// Library/Structures/WorkArea/RobotWorkArea
{attribute 'pack_mode' := '1'} 
// ------------------------------------------------------------------------- 
//  SRCI Robot Library                                                
// ------------------------------------------------------------------------- 
//                                                                           
//  Object:      RobotWorkArea                                       
//  Author:      Thorsten Brach                                                
//  Date:        2024-06-01
//
//  Description:                                              
//   
//                                                                           
//  Copyright: 
//    (C) 2024 Thorsten Brach. All rights reserved                                                                                                                                            
//             Licensed under the LGPL-3.0 license.
//                                                                           
//  Disclaimer:                                                                           
//    This project is provided without any guarantee and can be used for   
//    private and commercial purposes. Any use is at the user’s 
//    own risk and responsibility.
//
// -------------------------------------------------------------------------
TYPE RobotWorkArea :
STRUCT
  /// Timestamp
  Timestamp          : IEC_TIMESTAMP;
  /// Defines type of work area 
  AreaType           : AreaType;
  /// Defines violation condition 
  /// • FALSE (default) : Robot must not leave defined area
  /// • TRUE            : Robot must not enter defined area
  AreaMode           : BOOL := FALSE;
  /// Defines RC’s and robot’s behavior when robot violates work area 
  ReactionMode       : WorkAreaReactionMode;
  /// Specifies whether an active work area can be edited by function WriteWorkArea
  ///  TRUE            : Modification of active work area possible
  ///  FALSE (default) : Modification of active work areas not possible 
  ActiveModification : BOOL;
  /// Relates to AreaType Box, Cylinder and Sphere. 
  DefinitionMode     : DefinitionMode;
  /// Relates to AreaType Box, Cylinder and Sphere.
  /// Index of reference frame
  /// • 0: WCS (default)
  /// • 1..254: User frames 
  FrameNo            : USINT;
  /// Relates to AreaType Box, Cylinder and Sphere. 
  /// X-value of reference point in specified frame - Default: 0
  ZeroPointX         : REAL := 0;
  /// Relates to AreaType Box, Cylinder and Sphere. 
  /// Y-value of reference point in specified frame - Default: 0
  ZeroPointY         : REAL := 0;
  /// Relates to AreaType Box, Cylinder and Sphere. 
  /// Z-value of reference point in specified frame - Default: 0
  ZeroPointZ         : REAL := 0;
  /// Limit for cartesian X    
  X                  : RobotWorkAreaLimitCartesian;
  /// Limit for cartesian Y    
  Y                  : RobotWorkAreaLimitCartesian;
  /// Limit for cartesian Z    
  Z                  : RobotWorkAreaLimitCartesian;
  /// Relates to AreaType Sphere. 
  /// Radius of cylinder or sphere - Default 0
  Radius             : REAL := 0;
  /// Limits for Joint J1  
  J1Limit            : RobotWorkAreaLimitJoint;
  /// Limits for Joint J2  
  J2Limit            : RobotWorkAreaLimitJoint;
  /// Limits for Joint J3  
  J3Limit            : RobotWorkAreaLimitJoint;
  /// Limits for Joint J4  
  J4Limit            : RobotWorkAreaLimitJoint;
  /// Limits for Joint J5  
  J5Limit            : RobotWorkAreaLimitJoint;
  /// Limits for Joint J6  
  J6Limit            : RobotWorkAreaLimitJoint;
  /// Limits for Joint E1  
  E1Limit            : RobotWorkAreaLimitJoint;
  /// Limits for Joint E2  
  E2Limit            : RobotWorkAreaLimitJoint;
  /// Limits for Joint E3  
  E3Limit            : RobotWorkAreaLimitJoint;
  /// Limits for Joint E4  
  E4Limit            : RobotWorkAreaLimitJoint;
  /// Limits for Joint E5  
  E5Limit            : RobotWorkAreaLimitJoint;
  /// Limits for Joint E6  
  E6Limit            : RobotWorkAreaLimitJoint;
END_STRUCT
END_TYPE

// Library/Structures/WorkArea/RobotWorkAreaLimitCartesian
{attribute 'pack_mode' := '1'} 
// ------------------------------------------------------------------------- 
//  SRCI Robot Library                                                
// ------------------------------------------------------------------------- 
//                                                                           
//  Object:      RobotWorkAreaLimitCartesian                                       
//  Author:      Thorsten Brach                                                
//  Date:        2024-06-01
//
//  Description:                                              
//   
//                                                                           
//  Copyright: 
//    (C) 2024 Thorsten Brach. All rights reserved                                                                                                                                            
//             Licensed under the LGPL-3.0 license.
//                                                                           
//  Disclaimer:                                                                           
//    This project is provided without any guarantee and can be used for   
//    private and commercial purposes. Any use is at the user’s 
//    own risk and responsibility.
//
// -------------------------------------------------------------------------
TYPE RobotWorkAreaLimitCartesian :
STRUCT
  /// Relates to AreaType Box, Cylinder and Sphere. 
  /// Distance in negative Direction - Default 0  
  LowerLimit : REAL := 0;
  /// Relates to AreaType Box, Cylinder and Sphere.
  /// Distance in positive Direction - Default 0  
  UpperLimit : REAL := 0;
END_STRUCT
END_TYPE

// Library/Structures/WorkArea/RobotWorkAreaLimitJoint
{attribute 'pack_mode' := '1'} 
// ------------------------------------------------------------------------- 
//  SRCI Robot Library                                                
// ------------------------------------------------------------------------- 
//                                                                           
//  Object:      RobotWorkAreaLimitJoint                                       
//  Author:      Thorsten Brach                                                
//  Date:        2024-06-01
//
//  Description:                                              
//   
//                                                                           
//  Copyright: 
//    (C) 2024 Thorsten Brach. All rights reserved                                                                                                                                            
//             Licensed under the LGPL-3.0 license.
//                                                                           
//  Disclaimer:                                                                           
//    This project is provided without any guarantee and can be used for   
//    private and commercial purposes. Any use is at the user’s 
//    own risk and responsibility.
//
// -------------------------------------------------------------------------
TYPE RobotWorkAreaLimitJoint :
STRUCT
  /// Relates to AreaType Axes. 
  /// Negative work area limit for Joint
  /// • 0 (default) : No work area restriction of joint if lower and upper limit are set to 0  
  /// • 16#FFFF_FFFF: No lower work area restrictions for Joint
  LowerLimit : REAL := 0;
  /// Relates to AreaType Axes. 
  /// positive work area limit for Joint
  /// • 0 (default) : No work area restriction of joint if lower and upper limit of are set to 0  
  /// • 16#FFFF_FFFF: No lower work area restrictions for Joint
  UpperLimit : REAL := 0;  
END_STRUCT
END_TYPE

// Library/Structures/ExecutionModeAllowed
{attribute 'pack_mode' := '1'} 
// ------------------------------------------------------------------------- 
//  SRCI Robot Library                                                
// ------------------------------------------------------------------------- 
//                                                                           
//  Object:      ExecutionModeAllowed                                       
//  Author:      Thorsten Brach                                                
//  Date:        2024-06-01
//
//  Description:                                              
//   
//                                                                           
//  Copyright: 
//    (C) 2024 Thorsten Brach. All rights reserved                                                                                                                                            
//             Licensed under the LGPL-3.0 license.
//                                                                           
//  Disclaimer:                                                                           
//    This project is provided without any guarantee and can be used for   
//    private and commercial purposes. Any use is at the user’s 
//    own risk and responsibility.
//
// -------------------------------------------------------------------------
TYPE ExecutionModeAllowed :
STRUCT
  ///
  PRIMARY_SEQ         : BOOL;
  ///
  PRIMARY_SEQ_ABORT   : BOOL;
  ///
  SECONDARY_SEQ       : BOOL;
  ///
  SECONDARY_SEQ_ABORT : BOOL;
  ///
  PAR                 : BOOL := TRUE;
  ///
  PAR_TASK            : BOOL;
  ///
  PAR_TRIGGER         : BOOL;
  ///
  PAR_TRIGGER_TASK    : BOOL;
END_STRUCT
END_TYPE

// Library/Structures/MessageHeaderCommand
{attribute 'pack_mode' := '1'} 
// ------------------------------------------------------------------------- 
//  SRCI Robot Library                                                
// ------------------------------------------------------------------------- 
//                                                                           
//  Object:      MessageHeaderCommand                                       
//  Author:      Thorsten Brach                                                
//  Date:        2024-06-01
//
//  Description:                                              
//   
//                                                                           
//  Copyright: 
//    (C) 2024 Thorsten Brach. All rights reserved                                                                                                                                            
//             Licensed under the LGPL-3.0 license.
//                                                                           
//  Disclaimer:                                                                           
//    This project is provided without any guarantee and can be used for   
//    private and commercial purposes. Any use is at the user’s 
//    own risk and responsibility.
//
// -------------------------------------------------------------------------
TYPE MessageHeaderCommand :
STRUCT
  /// Byte 00-01 :  CMD type as per specification
  CmdType      : CmdType;
  /// Byte 02  : ExecutionMode (Bit 0..3)
  ExecMode     : BYTE;  
  /// Byte 03 : CMD priority (Bit 0..3)
  Prio         : BYTE;
  /// Byte 03 : Parameter Sequence (Bit 4..7 )
  ParSeq       : BYTE;
  /// Trigger related EmitterID
  EmitterID    : ARRAY[0..3] OF SINT;
  /// Trigger related ListenerID 
  ListenerID   : SINT;
  /// Reserved
  Reserved     : BYTE;
  //// Payload length defined by type per CMD definition. Processed by Appl. Layer Task.
  Payload      : ARRAY[0..RobotLibraryParameter.TELEGRAM_PAYLOAD_MAX] OF BYTE;  
END_STRUCT
END_TYPE

// Library/Structures/MessageHeaderResponse
{attribute 'pack_mode' := '1'} 
// ------------------------------------------------------------------------- 
//  SRCI Robot Library                                                
// ------------------------------------------------------------------------- 
//                                                                           
//  Object:      MessageHeaderResponse                                       
//  Author:      Thorsten Brach                                                
//  Date:        2024-06-01
//
//  Description:                                              
//   
//                                                                           
//  Copyright: 
//    (C) 2024 Thorsten Brach. All rights reserved                                                                                                                                            
//             Licensed under the LGPL-3.0 license.
//                                                                           
//  Disclaimer:                                                                           
//    This project is provided without any guarantee and can be used for   
//    private and commercial purposes. Any use is at the user’s 
//    own risk and responsibility.
//
// -------------------------------------------------------------------------
TYPE MessageHeaderResponse :
STRUCT
  /// Byte 03 : CMD priority (Bit 0..3)
  Prio                    : BYTE;
  /// Byte 03 : Parameter Sequence (Bit 4..7 )
  ParSeq                  : BYTE;
  /// Alarm Message Severity
  AlarmMessageSeverity    : Severity;
  /// Alarm Message Code
  AlarmMessageCode        : UINT;
  /// Number of Trigger based CMD invocations
  InvocationCounter       : USINT;
  /// Number of missed Triggers
  MissedInvocationCounter : USINT;
  /// FollowID of Trigger initiator
  OriginID                : WORD;
  /// RSP Payload defined by type per CMD definition. Generated by Appl. Layer Task
  Payload                 : ARRAY[0..RobotLibraryParameter.TELEGRAM_PAYLOAD_MAX] OF BYTE;  
END_STRUCT
END_TYPE

// Library/Constants/RobotLibraryConstants
{attribute 'qualified_only'}
// ------------------------------------------------------------------------- 
//  SRCI Robot Library                                                
// ------------------------------------------------------------------------- 
//                                                                           
//  Object:      RobotLibraryConstants                                       
//  Author:      Thorsten Brach                                                
//  Date:        2024-06-01
//
//  Description:                                              
//   
//                                                                           
//  Copyright: 
//    (C) 2024 Thorsten Brach. All rights reserved           
//             Licensed under the LGPL-3.0 license.                                                                                                                                 
//                                                                           
//  Disclaimer:                                                                           
//    This project is provided without any guarantee and can be used for   
//    private and commercial purposes. Any use is at the user’s 
//    own risk and responsibility.
//
// -------------------------------------------------------------------------
VAR_GLOBAL CONSTANT
  /// Minimal amount of tools
  TOOL_MIN             : DINT :=  16;
  /// Maximal amount of tools
  TOOL_MAX             : DINT := 255;
  /// Minimal amount of frames
  FRAME_MIN            : DINT :=  16;
  /// Maximal amount of frames
  FRAME_MAX            : DINT := 255;
  /// Minimal amount of loads
  LOAD_MIN             : DINT :=  16;  
  /// Maximal amount of loads
  LOAD_MAX             : DINT := 255;  
  /// Minimal amount of work areas
  WORK_AREAS_MIN       : DINT :=   8;  
  /// Maximal amount of work areas
  WORK_AREAS_MAX       : DINT := 255;  
  /// Maximal amount of bytes which are allowed to be exchanged with the sub program of the RC
  SUB_PROGRAM_DATA_MAX : DINT := 190;

  /// Version of SRCI specification
  /// Bit 0-4 : Minor version = Features        (0..31)
  /// Bit 5-7 : Major version = Breaking change (0..07)
  SRCIVersion            : VersionStruct := ( MajorVersion := 1, MinorVersion := 3, PatchVersion := 0);


  /// Minimal axes group ID
  AXES_GROUP_ID_MIN    : BYTE := 0;  
  /// Maximal axes groups ID
  AXES_GROUP_ID_MAX    : BYTE := 15;  



  /// OK = 0
  OK                   : DINT := 0;
  /// Running = 1
  RUNNING              : DINT := 1;
  /// Null pointer
  XNULL                : DWORD := 0;
  /// Null pointer
  NULL_POINTER         : POINTER TO BYTE := 0;
  
  /// Real conversion factor ( REAL * 100 -> TO_INT )
  REAL_CONVERSION_FACTOR  : REAL := 100;


  /// Active command
  ACTIVE_CMD           : UDINT := 1;
  /// Buffered command
  BUFFER_CMD           : UDINT := 2;
  
  /// Maximal length of additional text 
  MAX_ADD_TEXT_LENGTH  : DINT := 40; 
END_VAR

// Library/Constants/RobotLibraryDefines
{attribute 'qualified_only'}
VAR_GLOBAL
  /// Count of axes groups instances
  AxesGroupInstances : BYTE;
  /// Maximal length of type name
  MaxTypeNameLength  : INT;
END_VAR

// Library/Constants/RobotLibraryEvents
{attribute 'qualified_only'}
VAR_GLOBAL
  /// Program fault : Invalid step
  ERR_INVALID_STEP             : WORD := 1;
  /// Program fault : Invalid library parameter
  ERR_INVALID_LIBRARY_PARA     : WORD := 2;
  /// Program fault : Invalid axes groups ID
  ERR_INVALID_AXES_GROUP_ID    : WORD := 3;
  /// Program fault : Invalid amount of axes groups 
  ERR_INVALID_AXES_GROUP_COUNT : WORD := 4;
  
  ERR_FUNCTION_NOT_SUPPORTED   : WORD := 5;
  /// Program fault : Timeout during command execution 
  ERR_TIMEOUT_CMD              : WORD := 4;
END_VAR

// Library/Parameter/RobotLibraryParameter
{attribute 'qualified_only'}
// ------------------------------------------------------------------------- 
//  SRCI Robot Library                                                
// ------------------------------------------------------------------------- 
//                                                                           
//  Object:      Parameter                                       
//  Author:      Thorsten Brach                                                
//  Date:        2024-06-01
//
//  Description:                                              
//   
//                                                                           
//  Copyright: 
//    (C) 2024 Thorsten Brach. All rights reserved                                                                                                                                            
//             Licensed under the LGPL-3.0 license.
//                                                                           
//  Disclaimer:                                                                           
//    This project is provided without any guarantee and can be used for   
//    private and commercial purposes. Any use is at the user’s 
//    own risk and responsibility.
//
// -------------------------------------------------------------------------
VAR_GLOBAL CONSTANT
  /// Maximal amount of input data
  ROBOT_IN_DATA_MAX                   : UINT := 255;
  /// Maximal amount of output data
  ROBOT_OUT_DATA_MAX                  : UINT := 255;
  /// Maximal amount of tools
  TOOL_MAX                            : DINT := 16;
  /// Maximal amount of frames
  FRAME_MAX                           : DINT := 16;
  /// Maximal amount of loads
  LOAD_MAX                            : DINT := 16;  
  /// Maximal amount of work areas
  WORK_AREAS_MAX                      : DINT := 16;  
  /// Maximal amount of system logs
  SYSTEM_LOG_MAX                      : DINT := 32;  
  /// Maximal amount of message logs
  MESSAGE_LOG_MAX                     : DINT := 100;  
  /// Maximal amount of List entries 
  LIST_ENTRIES_MAX                    : DINT := 100;
  /// Maximal amount of bytes for the telegram payload
  TELEGRAM_PAYLOAD_MAX                : UDINT := 255;  
  /// Maximal amount of bytes for the parameter payload
  PARAMETER_PAYLOAD_MAX               : DINT := 128;  
  /// Maximal amount of bytes for the response payload
  RESPONSE_PAYLOAD_MAX                : DINT := 128;  
  /// Maximal amount of bytes that can be exchanged with the sub program on the RC
  SUB_PROGRAM_DATA_MAX                : DINT := 189;
  /// Maximal amount of spline data
  SPLINE_DATA_MAX                     : DINT := 64;
  /// Maximal amount of entries in the Active Command Register
  ACTIVE_CMD_REGISTER_ENTRIES_MAX     : DINT := 50;
  /// Maximal amount of message codes
  MESSAGE_CODES_MAX                   : DINT := 15;
  /// Maximal amount of fragments
  FRAGMENT_MAX                        : DINT := 9;
  /// Use two sequences in telegram ?
  TWO_SEQUENCES                       : BOOL := FALSE; 
  /// Flag to indicate that the byte order must be changed
  SWAP_BYTE_ORDER                     : BOOL := TRUE; 
  /// Life Sign Timeout
  LIFE_SIGN_TIMEOUT                   : TIME := T#40MS;
  /// Timeout for checking for invalid frames
  INVALID_FRAMES_CHECK_TIMEOUT        : TIME := T#60S;
END_VAR

// Library/Functions/Common/CheckTimeout
FUNCTION CheckTimeout : DINT
// ------------------------------------------------------------------------- 
//  SRCI Robot Library                                                
// ------------------------------------------------------------------------- 
//                                                                           
//  Object:      SwapBytes                                       
//  Author:      Thorsten Brach                                                
//  Date:        2024-12-18
//
//  Description:                                              
//   
//                                                                           
//  Copyright: 
//    (C) 2024 Thorsten Brach. All rights reserved                                                                                                                                            
//             Licensed under the LGPL-3.0 license.
//                                                                           
//  Disclaimer:                                                                           
//    This project is provided without any guarantee and can be used for   
//    private and commercial purposes. Any use is at the user’s 
//    own risk and responsibility.
//
// -------------------------------------------------------------------------
VAR_INPUT
  /// Reference to TON instance
  rTimer : REFERENCE TO TON;
END_VAR

// Call timer 
rTimer();

// check if timer elapsed
IF (rTimer.Q = TRUE)
THEN
  // assign return value
  CheckTimeout := RobotLibraryConstants.OK;
ELSE
  // assign return value
  CheckTimeout := RobotLibraryConstants.RUNNING;
END_IF

END_FUNCTION

// Library/Functions/Swap/SwapBytes
FUNCTION SwapBytes 
// ------------------------------------------------------------------------- 
//  SRCI Robot Library                                                
// ------------------------------------------------------------------------- 
//                                                                           
//  Object:      SwapBytes                                       
//  Author:      Thorsten Brach                                                
//  Date:        2024-06-01
//
//  Description:                                              
//   
//                                                                           
//  Copyright: 
//    (C) 2024 Thorsten Brach. All rights reserved                                                                                                                                            
//             Licensed under the LGPL-3.0 license.
//                                                                           
//  Disclaimer:                                                                           
//    This project is provided without any guarantee and can be used for   
//    private and commercial purposes. Any use is at the user’s 
//    own risk and responsibility.
//
// -------------------------------------------------------------------------
VAR_INPUT
  /// pointer to data type
  pValue : POINTER TO BYTE;
  /// size of data type
  Size  : UDINT;
END_VAR

VAR
  /// Pointer to low word low byte
  _pLwLb    : POINTER TO BYTE;
  /// Pointer to low word high byte
  _pLwHb    : POINTER TO BYTE;
  /// Pointer to high word low byte
  _pHwLb    : POINTER TO BYTE;
  /// Pointer to high word high byte
  _pHwHb    : POINTER TO BYTE;  
   /// temporary bytes
  _tmpBytes : ARRAY[1..4] OF BYTE;  
END_VAR

IF ( RobotLibraryParameter.SWAP_BYTE_ORDER AND Size = 2)
THEN
 _pLwLb := pValue + 0;
 _pLwHb := pValue + 1;
  
  // swap bytes
 _tmpBytes[1] := _pLwHb^;
 _tmpBytes[2] := _pLwLb^;
  
  // copy bytes to data type
  SysDepMemCpy(pDest := pValue, pSrc := ADR(_tmpBytes), DataLen := Size);
END_IF


IF ( RobotLibraryParameter.SWAP_BYTE_ORDER AND Size = 4)
THEN
 _pLwLb := pValue + 0;
 _pLwHb := pValue + 1;
 _pHwLb := pValue + 2;
 _pHwHb := pValue + 3;
  
  // swap bytes
 _tmpBytes[1] := _pHwHb^;
 _tmpBytes[2] := _pHwLb^;
 _tmpBytes[3] := _pLwHb^;
 _tmpBytes[4] := _pLwLb^;
  
  // copy bytes to data type
  SysDepMemCpy( pDest := pValue, pSrc := ADR(_tmpBytes), DataLen := Size);  
END_IF

END_FUNCTION

// Library/Functions/Common/SetTimeout
FUNCTION SetTimeout : DINT
// ------------------------------------------------------------------------- 
//  SRCI Robot Library                                                
// ------------------------------------------------------------------------- 
//                                                                           
//  Object:      SwapBytes                                       
//  Author:      Thorsten Brach                                                
//  Date:        2024-12-18
//
//  Description:                                              
//   
//                                                                           
//  Copyright: 
//    (C) 2024 Thorsten Brach. All rights reserved                                                                                                                                            
//             Licensed under the LGPL-3.0 license.
//                                                                           
//  Disclaimer:                                                                           
//    This project is provided without any guarantee and can be used for   
//    private and commercial purposes. Any use is at the user’s 
//    own risk and responsibility.
//
// -------------------------------------------------------------------------
VAR_INPUT
  /// Timeout to be set
  PT     : TIME;
  /// Reference to TON instance
  rTimer : REFERENCE TO TON;
END_VAR

rTimer(IN := FALSE);          // Reset timer
rTimer(PT := PT, IN := TRUE); // Start timer

// assign return value
SetTimeout := RobotLibraryConstants.OK;

END_FUNCTION

// Library/Functions/Convert/DT/DATE_TO_IEC_DATE
FUNCTION DATE_TO_IEC_DATE : IEC_DATE
// ------------------------------------------------------------------------- 
//  SRCI Robot Library                                                
// ------------------------------------------------------------------------- 
//                                                                           
//  Object:      DATE_TO_IEC_DATE                                       
//  Author:      Thorsten Brach                                                
//  Date:        2024-06-01
//
//  Description:                                              
//   
//                                                                           
//  Copyright: 
//    (C) 2024 Thorsten Brach. All rights reserved                                                                                                                                            
//             Licensed under the LGPL-3.0 license.
//                                                                           
//  Disclaimer:                                                                           
//    This project is provided without any guarantee and can be used for   
//    private and commercial purposes. Any use is at the user’s 
//    own risk and responsibility.
//
// -------------------------------------------------------------------------
VAR_INPUT
  Value    : DATE;
END_VAR

VAR
 _tmpDate1 : DWORD;
 _tmpDate2 : DWORD;
 _initDate : DATE := DATE#1990-01-01;
 END_VAR

// Siemens Dateformat is Day since 01.01.1990
// TwinCat Dateformat is seconds sinde 01.01.1970
// Calculation : 
// ( [TwinCat current date] - [ TwinCat 01.01.1970] ) / [Seconds a Day] = Days sinde 01.01.1990 (Siemens Format)

// copy date to dword
SysDepMemCpy( pDest := ADR(_tmpDate1), pSrc := ADR( Value   ), DataLen := SIZEOF( Value   ));
// copy date to dword
SysDepMemCpy( pDest := ADR(_tmpDate2), pSrc := ADR(_initDate), DataLen := SIZEOF(_initDate));

// calculate IEC Date :  
DATE_TO_IEC_DATE := UDINT_TO_UINT((_tmpDate1 - _tmpDate2) / 86400); // 86400 Seconds = 1 day

END_FUNCTION

// Library/Functions/Convert/DT/IEC_DATE_TO_DATE
FUNCTION IEC_DATE_TO_DATE : DATE
// ------------------------------------------------------------------------- 
//  SRCI Robot Library                                                
// ------------------------------------------------------------------------- 
//                                                                           
//  Object:      IEC_DATE_TO_DATE                                       
//  Author:      Thorsten Brach                                                
//  Date:        2025-01-05
//
//  Description:                                              
//   
//                                                                           
//  Copyright: 
//    (C) 2025 Thorsten Brach. All rights reserved                                                                                                                                            
//             Licensed under the LGPL-3.0 license.
//                                                                           
//  Disclaimer:                                                                           
//    This project is provided without any guarantee and can be used for   
//    private and commercial purposes. Any use is at the user’s 
//    own risk and responsibility.
//
// -------------------------------------------------------------------------
VAR_INPUT
  Value    : IEC_DATE;
END_VAR

VAR
 _tmpDate1 : DWORD;
 _initDate : DATE := DATE#1990-01-01;
 END_VAR

// Siemens Dateformat is Day since 01.01.1990
// TwinCat Dateformat is seconds sinde 01.01.1970
// Calculation : 
// ( [ TwinCat 01.01.1990] + [IEC Date]) * [Seconds a Day] = (TwinCat Format)

// copy date to dword
SysDepMemCpy( pDest := ADR(_tmpDate1), pSrc := ADR( _initDate ), DataLen := SIZEOF( _initDate ));

// calculate IEC Date :  
IEC_DATE_TO_DATE := DWORD_TO_DATE( _tmpDate1 + ( Value * 86400)); // 86400 Seconds = 1 day

END_FUNCTION

// Library/Functions/Convert/DT/IEC_TIME_TO_TIME
FUNCTION IEC_TIME_TO_TIME : TOD
// ------------------------------------------------------------------------- 
//  SRCI Robot Library                                                
// ------------------------------------------------------------------------- 
//                                                                           
//  Object:      IEC_TIME_TO_TIME                                       
//  Author:      Thorsten Brach                                                
//  Date:        2025-01-05
//
//  Description:                                              
//   
//                                                                           
//  Copyright: 
//    (C) 2025 Thorsten Brach. All rights reserved                                                                                                                                            
//             Licensed under the LGPL-3.0 license.
//                                                                           
//  Disclaimer:                                                                           
//    This project is provided without any guarantee and can be used for   
//    private and commercial purposes. Any use is at the user’s 
//    own risk and responsibility.
//
// -------------------------------------------------------------------------
VAR_INPUT
  Value : IEC_TIME;
END_VAR

IEC_TIME_TO_TIME := Value;

END_FUNCTION

// Library/Functions/Convert/DT/IEC_TIMESTAMP_TO_DT
FUNCTION IEC_TIMESTAMP_TO_DT : DT
// ------------------------------------------------------------------------- 
//  SRCI Robot Library                                                
// ------------------------------------------------------------------------- 
//                                                                           
//  Object:      TIME_TO_IEC_TIME                                       
//  Author:      Thorsten Brach                                                
//  Date:        2025-01-05
//
//  Description:                                              
//   
//                                                                           
//  Copyright: 
//    (C) 2025 Thorsten Brach. All rights reserved                                                                                                                                            
//             Licensed under the LGPL-3.0 license.
//                                                                           
//  Disclaimer:                                                                           
//    This project is provided without any guarantee and can be used for   
//    private and commercial purposes. Any use is at the user’s 
//    own risk and responsibility.
//
// -------------------------------------------------------------------------
VAR_INPUT
  Value : IEC_TIMESTAMP;
END_VAR

VAR
  /// internal date
 _date    : DATE;
  /// internal date as string
 _dateStr : STRING;
  /// internal time
 _time    : TOD;
  /// internal time as string
 _timeStr : STRING;
END_VAR

_date := IEC_DATE_TO_DATE(Value.IEC_DATE); 
_time := IEC_TIME_TO_TIME(Value.IEC_TIME); 


// Example : DATE#2025-1-5
_dateStr := DATE_TO_STRING(_date);
// Example : DT#2025-1-5
_dateStr := strReplace(_dateStr, 'D#', 'DT#');

// Example : TOD#15:18:4.567
_timeStr :=  TOD_TO_STRING(_time);
// Example : -15:18:4.567
_timeStr := strReplace(_timeStr, 'TOD#', '-');

// Example : DT#2025-1-5-15:18:4.567
IEC_TIMESTAMP_TO_DT := STRING_TO_DT( Concat(_dateStr,_timeStr));

END_FUNCTION

// Library/Functions/String/StrReplace
/// Returns a given string where a given substing is replaced by another substring
FUNCTION StrReplace : STRING(255)
// ------------------------------------------------------------------------- 
//  SRCI Robot Library                                                
// ------------------------------------------------------------------------- 
//                                                                           
//  Object:      SwapBytes                                       
//  Author:      Thorsten Brach                                                
//  Date:        2024-12-18
//
//  Description:                                              
//   
//                                                                           
//  Copyright: 
//    (C) 2024 Thorsten Brach. All rights reserved                                                                                                                                            
//             Licensed under the LGPL-3.0 license.
//                                                                           
//  Disclaimer:                                                                           
//    This project is provided without any guarantee and can be used for   
//    private and commercial purposes. Any use is at the user’s 
//    own risk and responsibility.
//
// -------------------------------------------------------------------------
VAR_INPUT
  /// content string
  Str      : STRING(255);
  /// sub string with the old characters
  SubStr1  : STRING(255);
  /// sub string with the new characters
  SubStr2  : STRING(255);
END_VAR

WHILE (FIND(Str, SubStr1) > 0)
DO  
  Str := Replace(Str, SubStr2, LEN(SubStr1), FIND(Str, SubStr1)); 
END_WHILE

StrReplace := Str;

END_FUNCTION

// Library/Functions/Convert/DT/TIME_TO_IEC_TIME
FUNCTION TIME_TO_IEC_TIME : IEC_TIME
// ------------------------------------------------------------------------- 
//  SRCI Robot Library                                                
// ------------------------------------------------------------------------- 
//                                                                           
//  Object:      TIME_TO_IEC_TIME                                       
//  Author:      Thorsten Brach                                                
//  Date:        2024-06-01
//
//  Description:                                              
//   
//                                                                           
//  Copyright: 
//    (C) 2024 Thorsten Brach. All rights reserved                                                                                                                                            
//             Licensed under the LGPL-3.0 license.
//                                                                           
//  Disclaimer:                                                                           
//    This project is provided without any guarantee and can be used for   
//    private and commercial purposes. Any use is at the user’s 
//    own risk and responsibility.
//
// -------------------------------------------------------------------------
VAR_INPUT
  Value : TOD;
END_VAR

TIME_TO_IEC_TIME := Value;

END_FUNCTION

// Library/Functions/Convert/Misc/ArmConfigParameterToBytes
FUNCTION ArmConfigParameterToBytes : ARRAY[0..1] of BYTE
// ------------------------------------------------------------------------- 
//  SRCI Robot Library                                                
// ------------------------------------------------------------------------- 
//                                                                           
//  Object:      ArmConfigParameterToBytes                                       
//  Author:      Thorsten Brach                                                
//  Date:        2025-01-30
//
//  Description:                                              
//   
//                                                                           
//  Copyright: 
//    (C) 2025 Thorsten Brach. All rights reserved                                                                                                                                            
//             Licensed under the LGPL-3.0 license.
//                                                                           
//  Disclaimer:                                                                           
//    This project is provided without any guarantee and can be used for   
//    private and commercial purposes. Any use is at the user’s 
//    own risk and responsibility.
//
// -------------------------------------------------------------------------
VAR_INPUT
 /// ArmConfigParameter
 Value: ArmConfigParameter;
END_VAR

ArmConfigParameterToBytes[0].0 := Value.Shoulder.0;
ArmConfigParameterToBytes[0].1 := Value.Shoulder.1;
ArmConfigParameterToBytes[0].2 := Value.Shoulder.2;
ArmConfigParameterToBytes[0].3 := Value.Shoulder.3;
ArmConfigParameterToBytes[0].4 := Value.Elbow.0;
ArmConfigParameterToBytes[0].5 := Value.Elbow.1;
ArmConfigParameterToBytes[0].6 := Value.Elbow.2;
ArmConfigParameterToBytes[0].7 := Value.Elbow.3;
ArmConfigParameterToBytes[1].0 := Value.Wrist.0;
ArmConfigParameterToBytes[1].1 := Value.Wrist.1;
ArmConfigParameterToBytes[1].2 := Value.Wrist.2;
ArmConfigParameterToBytes[1].3 := Value.Wrist.3;
ArmConfigParameterToBytes[1].4 := FALSE;
ArmConfigParameterToBytes[1].5 := FALSE;
ArmConfigParameterToBytes[1].6 := FALSE;
ArmConfigParameterToBytes[1].7 := FALSE;

END_FUNCTION

// Library/Functions/Convert/Misc/BytesToRCSupportedFunctions
FUNCTION BytesToRCSupportedFunctions : RCSupportedFunctions
// ------------------------------------------------------------------------- 
//  SRCI Robot Library                                                
// ------------------------------------------------------------------------- 
//                                                                           
//  Object:      BytesToRCSupportedFunctions                                       
//  Author:      Thorsten Brach                                                
//  Date:        2024-12-18
//
//  Description:                                              
//   
//                                                                           
//  Copyright: 
//    (C) 2024 Thorsten Brach. All rights reserved                                                                                                                                            
//             Licensed under the LGPL-3.0 license.
//                                                                           
//  Disclaimer:                                                                           
//    This project is provided without any guarantee and can be used for   
//    private and commercial purposes. Any use is at the user’s 
//    own risk and responsibility.
//
// -------------------------------------------------------------------------
VAR_INPUT
  Bytes : ARRAY [0..18] OF BYTE;
END_VAR

// Byte 00 - Bit 0  
BytesToRCSupportedFunctions.Reserved                   := Bytes[00].0;
// Byte 00 - Bit 1 
BytesToRCSupportedFunctions.ReadRobotData              := Bytes[00].1;
// Byte 00 - Bit 2  
BytesToRCSupportedFunctions.EnableRobot                := Bytes[00].2;
// Byte 00 - Bit 3  
BytesToRCSupportedFunctions.GroupReset                 := Bytes[00].3;
// Byte 00 - Bit 4  
BytesToRCSupportedFunctions.ReadActualPosition         := Bytes[00].4;
// Byte 00 - Bit 5 
BytesToRCSupportedFunctions.ReadActualPositionCyclic   := Bytes[00].5;
// Byte 00 - Bit 6  
BytesToRCSupportedFunctions.ExchangeConfiguration      := Bytes[00].6;
// Byte 00 - Bit 7  
BytesToRCSupportedFunctions.SetSequence                := Bytes[00].7;

// Byte 01 - Bit 0  
BytesToRCSupportedFunctions.ChangeSpeedOverride        := Bytes[01].0;
// Byte 01 - Bit 1  
BytesToRCSupportedFunctions.ReadMessages               := Bytes[01].1;
// Byte 01 - Bit 2  
BytesToRCSupportedFunctions.ReadRobotReferenceDynamics := Bytes[01].2;
// Byte 01 - Bit 3  
BytesToRCSupportedFunctions.WriteFrameData             := Bytes[01].3;
// Byte 01 - Bit 4  
BytesToRCSupportedFunctions.WriteToolData              := Bytes[01].4;
// Byte 01 - Bit 5  
BytesToRCSupportedFunctions.WriteLoadData              := Bytes[01].5;
// Byte 01 - Bit 6  
BytesToRCSupportedFunctions.WriteRobotReferenceDynamics:= Bytes[01].6;
// Byte 01 - Bit 7  
BytesToRCSupportedFunctions.WriteRobotDefaultDynamics  := Bytes[01].7;

// Byte 02 - Bit 0  
BytesToRCSupportedFunctions.ReadRobotDefaultDynamics   := Bytes[02].0;
// Byte 02 - Bit 1  
BytesToRCSupportedFunctions.ReadFrameData              := Bytes[02].1;
// Byte 02 - Bit 2  
BytesToRCSupportedFunctions.ReadToolData               := Bytes[02].2;
// Byte 02 - Bit 3  
BytesToRCSupportedFunctions.ReadLoadData               := Bytes[02].3;
// Byte 02 - Bit 4  
BytesToRCSupportedFunctions.ReadRobotSWLimits          := Bytes[02].4;
// Byte 02 - Bit 5  
BytesToRCSupportedFunctions.GroupJog                   := Bytes[02].5;
// Byte 02 - Bit 6  
BytesToRCSupportedFunctions.MoveLinearAbsolute         := Bytes[02].6;
// Byte 02 - Bit 7  
BytesToRCSupportedFunctions.MoveDirectAbsolute         := Bytes[02].7;

// Byte 03 - Bit 0  
BytesToRCSupportedFunctions.MoveAxesAbsolute           := Bytes[03].0;
// Byte 03 - Bit 1  
BytesToRCSupportedFunctions.GroupStop                  := Bytes[03].1;
// Byte 03 - Bit 2
BytesToRCSupportedFunctions.GroupContinue              := Bytes[03].2;
// Byte 03 - Bit 3
BytesToRCSupportedFunctions.GroupInterrupt             := Bytes[03].3;
// Byte 03 - Bit 4
BytesToRCSupportedFunctions.ReturnToPrimary            := Bytes[03].4;
// Byte 03 - Bit 5
BytesToRCSupportedFunctions.MoveLinearAbsoluteJ        := Bytes[03].5;
// Byte 03 - Bit 6
BytesToRCSupportedFunctions.MoveDirectRelative         := Bytes[03].6;
// Byte 03 - Bit 7
BytesToRCSupportedFunctions.MoveAxesRelative           := Bytes[03].7;

// Byte 04 - Bit 0
BytesToRCSupportedFunctions.MoveCircularAbsolute       := Bytes[04].0;
// Byte 04 - Bit 1
BytesToRCSupportedFunctions.MoveCircularRelative       := Bytes[04].1;
// Byte 04 - Bit 2
BytesToRCSupportedFunctions.MoveLinearOffset           := Bytes[04].2;
// Byte 04 - Bit 3
BytesToRCSupportedFunctions.MoveDirectOffset           := Bytes[04].3;
// Byte 04 - Bit 4
BytesToRCSupportedFunctions.WaitTime                   := Bytes[04].4;
// Byte 04 - Bit 5
BytesToRCSupportedFunctions.ReadDigitalInputs          := Bytes[04].5;
// Byte 04 - Bit 6
BytesToRCSupportedFunctions.ReadDigitalOutputs         := Bytes[04].6;
// Byte 04 - Bit 7
BytesToRCSupportedFunctions.WriteDigitalOutputs        := Bytes[04].7;

// Byte 05 - Bit 0
BytesToRCSupportedFunctions.ReadIntegers               := Bytes[05].0;
// Byte 05 - Bit 1
BytesToRCSupportedFunctions.ReadReals                  := Bytes[05].1;
// Byte 05 - Bit 2
BytesToRCSupportedFunctions.WriteIntegers              := Bytes[05].2;
// Byte 05 - Bit 3
BytesToRCSupportedFunctions.WriteReals                 := Bytes[05].3;
// Byte 05 - Bit 4
BytesToRCSupportedFunctions.MoveLinearCam              := Bytes[05].4;
// Byte 05 - Bit 5
BytesToRCSupportedFunctions.MoveDirectCam              := Bytes[05].5;
// Byte 05 - Bit 6
BytesToRCSupportedFunctions.MoveCircularCam            := Bytes[05].6;
// Byte 05 - Bit 7
BytesToRCSupportedFunctions.SetTriggerRegister         := Bytes[05].7;

// Byte 06 - Bit 0
BytesToRCSupportedFunctions.SetTriggerLimit            := Bytes[06].0;
// Byte 06 - Bit 1
BytesToRCSupportedFunctions.SetTriggerUser             := Bytes[06].1;
// Byte 06 - Bit 2
BytesToRCSupportedFunctions.SetTriggerError            := Bytes[06].2;
// Byte 06 - Bit 3
BytesToRCSupportedFunctions.ReactAtTrigger             := Bytes[06].3;
// Byte 06 - Bit 4
BytesToRCSupportedFunctions.WaitForTrigger             := Bytes[06].4;
// Byte 06 - Bit 5
BytesToRCSupportedFunctions.ReadSystemVariable         := Bytes[06].5;
// Byte 06 - Bit 6
BytesToRCSupportedFunctions.WriteSystemVariable        := Bytes[06].6;
// Byte 06 - Bit 7
BytesToRCSupportedFunctions.CalculateForwardKinematic  := Bytes[06].7;

// Byte 07 - Bit 0
BytesToRCSupportedFunctions.CalculateInverseKinematic  := Bytes[07].0;
// Byte 07 - Bit 1
BytesToRCSupportedFunctions.CalculateCartesianPosition := Bytes[07].1;
// Byte 07 - Bit 2
BytesToRCSupportedFunctions.CalculateTool              := Bytes[07].2;
// Byte 07 - Bit 3
BytesToRCSupportedFunctions.CalculateFrame             := Bytes[07].3;
// Byte 07 - Bit 4
BytesToRCSupportedFunctions.ActivateNextCommand        := Bytes[07].4;
// Byte 07 - Bit 5
BytesToRCSupportedFunctions.ShiftPosition              := Bytes[07].5;
// Byte 07 - Bit 6
BytesToRCSupportedFunctions.CallSubprogram             := Bytes[07].6;
// Byte 07 - Bit 7
BytesToRCSupportedFunctions.MoveLinearRelative         := Bytes[07].7;

// Byte 08 - Bit 0
BytesToRCSupportedFunctions.WriteCallSubprogramCyclic  := Bytes[08].0;
// Byte 08 - Bit 1
BytesToRCSupportedFunctions.ReadCallSubprogramCyclic   := Bytes[08].1;
// Byte 08 - Bit 2
BytesToRCSupportedFunctions.StopSubprogram             := Bytes[08].2;
// Byte 08 - Bit 3
BytesToRCSupportedFunctions.ReadDHParameter            := Bytes[08].3;
// Byte 08 - Bit 4
BytesToRCSupportedFunctions.RestartController          := Bytes[08].4;
// Byte 08 - Bit 5
BytesToRCSupportedFunctions.ReadActualTCPVelocity      := Bytes[08].5;
// Byte 08 - Bit 6
BytesToRCSupportedFunctions.UserLogin                  := Bytes[08].6;
// Byte 08 - Bit 7
BytesToRCSupportedFunctions.SwitchLanguage             := Bytes[08].7;

// Byte 09 - Bit 0
BytesToRCSupportedFunctions.WriteRobotSWLimits         := Bytes[09].0;
// Byte 09 - Bit 1
BytesToRCSupportedFunctions.SetOperationMode           := Bytes[09].1;
// Byte 09 - Bit 2
BytesToRCSupportedFunctions.ReadWorkArea               := Bytes[09].2;
// Byte 09 - Bit 3
BytesToRCSupportedFunctions.WriteWorkArea              := Bytes[09].3;
// Byte 09 - Bit 4
BytesToRCSupportedFunctions.ActivateWorkArea           := Bytes[09].4;
// Byte 09 - Bit 5
BytesToRCSupportedFunctions.MonitorWorkArea            := Bytes[09].5;
// Byte 09 - Bit 6
BytesToRCSupportedFunctions.MoveApproachLinear         := Bytes[09].6;
// Byte 09 - Bit 7
BytesToRCSupportedFunctions.MoveDepartLinear           := Bytes[09].7;

// Byte 10 - Bit 0
BytesToRCSupportedFunctions.MoveApproachDirect         := Bytes[10].0;
// Byte 10 - Bit 1
BytesToRCSupportedFunctions.MoveDepartDirect           := Bytes[10].1;
// Byte 10 - Bit 2
BytesToRCSupportedFunctions.SearchHardstop             := Bytes[10].2;
// Byte 10 - Bit 3
BytesToRCSupportedFunctions.SearchHardstopJ            := Bytes[10].3;
// Byte 10 - Bit 4
BytesToRCSupportedFunctions.MovePickPlaceLinear        := Bytes[10].4;
// Byte 10 - Bit 5
BytesToRCSupportedFunctions.MovePickPlaceDirect        := Bytes[10].5;
// Byte 10 - Bit 6
BytesToRCSupportedFunctions.ActivateConveyorTracking   := Bytes[10].6;
// Byte 10 - Bit 7
BytesToRCSupportedFunctions.RedefineTrackingPosition   := Bytes[10].7;

// Byte 11 - Bit 0
BytesToRCSupportedFunctions.SyncToConveyor             := Bytes[11].0;
// Byte 11 - Bit 1
BytesToRCSupportedFunctions.ConfigureConveyor          := Bytes[11].1;
// Byte 11 - Bit 2
BytesToRCSupportedFunctions.MoveSuperImposed           := Bytes[11].2;
// Byte 11 - Bit 3
BytesToRCSupportedFunctions.MoveSuperImposedDynamic    := Bytes[11].3;
// Byte 11 - Bit 4
BytesToRCSupportedFunctions.ReadAnalogInput            := Bytes[11].4;
// Byte 11 - Bit 5
BytesToRCSupportedFunctions.ReadAnalogOutput           := Bytes[11].5;
// Byte 11 - Bit 6
BytesToRCSupportedFunctions.WriteAnalogOutput          := Bytes[11].6;
// Byte 11 - Bit 7
BytesToRCSupportedFunctions.MeasuringInput             := Bytes[11].7;

// Byte 12 - Bit 0
BytesToRCSupportedFunctions.AbortMeasuringInput        := Bytes[12].0;
// Byte 12 - Bit 1
BytesToRCSupportedFunctions.SetTriggerMotion           := Bytes[12].1;
// Byte 12 - Bit 2
BytesToRCSupportedFunctions.OpenBrake                  := Bytes[12].2;
// Byte 12 - Bit 3
BytesToRCSupportedFunctions.PathAccuracyMode           := Bytes[12].3;
// Byte 12 - Bit 4
BytesToRCSupportedFunctions.AvoidSingularity           := Bytes[12].4;
// Byte 12 - Bit 5
BytesToRCSupportedFunctions.ForceControl               := Bytes[12].5;
// Byte 12 - Bit 6
BytesToRCSupportedFunctions.ForceLimit                 := Bytes[12].6;
// Byte 12 - Bit 7
BytesToRCSupportedFunctions.ReadActualForce            := Bytes[12].7;

// Byte 13 - Bit 0
BytesToRCSupportedFunctions.BrakeTest                  := Bytes[13].0;
// Byte 13 - Bit 1
BytesToRCSupportedFunctions.SoftSwitchTCP              := Bytes[13].1;
// Byte 13 - Bit 2
BytesToRCSupportedFunctions.CreateSpline               := Bytes[13].2;
// Byte 13 - Bit 3
BytesToRCSupportedFunctions.DeleteSpline               := Bytes[13].3;
// Byte 13 - Bit 4
BytesToRCSupportedFunctions.MoveSpline                 := Bytes[13].4;
// Byte 13 - Bit 5
BytesToRCSupportedFunctions.DynamicSpline              := Bytes[13].5;
// Byte 13 - Bit 6
BytesToRCSupportedFunctions.LoadMeasurementAutomatic   := Bytes[13].6;
// Byte 13 - Bit 7
BytesToRCSupportedFunctions.LoadMeasurementSequential  := Bytes[13].7;

// Byte 14 - Bit 0
BytesToRCSupportedFunctions.CollisionDetection         := Bytes[14].0;
// Byte 14 - Bit 1
BytesToRCSupportedFunctions.FreeDrive                  := Bytes[14].1;
// Byte 14 - Bit 2
BytesToRCSupportedFunctions.UnitMeasurement            := Bytes[14].2;
// Byte 14 - Bit 3
BytesToRCSupportedFunctions.Byte14Bit03                := Bytes[14].3;
// Byte 14 - Bit 4
BytesToRCSupportedFunctions.Byte14Bit04                := Bytes[14].4;
// Byte 14 - Bit 5
BytesToRCSupportedFunctions.Byte14Bit05                := Bytes[14].5;
// Byte 14 - Bit 6
BytesToRCSupportedFunctions.Byte14Bit06                := Bytes[14].6;
// Byte 14 - Bit 7
BytesToRCSupportedFunctions.Byte14Bit07                := Bytes[14].7;

// Byte 15 - Bit 0
BytesToRCSupportedFunctions.Byte15Bit00                := Bytes[15].0;
// Byte 15 - Bit 1
BytesToRCSupportedFunctions.Byte15Bit01                := Bytes[15].1;
// Byte 15 - Bit 2
BytesToRCSupportedFunctions.Byte15Bit02                := Bytes[15].2;
// Byte 15 - Bit 3
BytesToRCSupportedFunctions.Byte15Bit03                := Bytes[15].3;
// Byte 15 - Bit 4
BytesToRCSupportedFunctions.Byte15Bit04                := Bytes[15].4;
// Byte 15 - Bit 5
BytesToRCSupportedFunctions.Byte15Bit05                := Bytes[15].5;
// Byte 15 - Bit 6
BytesToRCSupportedFunctions.Byte15Bit06                := Bytes[15].6;
// Byte 15 - Bit 7
BytesToRCSupportedFunctions.Byte15Bit07                := Bytes[15].7;

// Byte 16 - Bit 0
BytesToRCSupportedFunctions.Byte16Bit00                := Bytes[16].0;
// Byte 15 - Bit 1
BytesToRCSupportedFunctions.Byte16Bit01                := Bytes[16].1;
// Byte 15 - Bit 2
BytesToRCSupportedFunctions.Byte16Bit02                := Bytes[16].2;
// Byte 15 - Bit 3
BytesToRCSupportedFunctions.Byte16Bit03                := Bytes[16].3;
// Byte 15 - Bit 4
BytesToRCSupportedFunctions.Byte16Bit04                := Bytes[16].4;
// Byte 15 - Bit 5
BytesToRCSupportedFunctions.Byte16Bit05                := Bytes[16].5;
// Byte 15 - Bit 6
BytesToRCSupportedFunctions.Byte16Bit06                := Bytes[16].6;
// Byte 15 - Bit 7
BytesToRCSupportedFunctions.Byte16Bit07                := Bytes[16].7;

// Byte 17 - Bit 0
BytesToRCSupportedFunctions.Byte17Bit00                := Bytes[17].0;
// Byte 17 - Bit 1
BytesToRCSupportedFunctions.Byte17Bit01                := Bytes[17].1;
// Byte 17 - Bit 2
BytesToRCSupportedFunctions.Byte17Bit02                := Bytes[17].2;
// Byte 17 - Bit 3
BytesToRCSupportedFunctions.Byte17Bit03                := Bytes[17].3;
// Byte 17 - Bit 4
BytesToRCSupportedFunctions.Byte17Bit04                := Bytes[17].4;
// Byte 17 - Bit 5
BytesToRCSupportedFunctions.Byte17Bit05                := Bytes[17].5;
// Byte 17 - Bit 6
BytesToRCSupportedFunctions.Byte17Bit06                := Bytes[17].6;
// Byte 17 - Bit 7
BytesToRCSupportedFunctions.Byte17Bit07                := Bytes[17].7;

// Byte 18 - Bit 0
BytesToRCSupportedFunctions.Byte18Bit00                := Bytes[18].0;
// Byte 18 - Bit 1
BytesToRCSupportedFunctions.Byte18Bit01                := Bytes[18].1;
// Byte 18 - Bit 2
BytesToRCSupportedFunctions.Byte18Bit02                := Bytes[18].2;
// Byte 18 - Bit 3
BytesToRCSupportedFunctions.Byte18Bit03                := Bytes[18].3;
// Byte 18 - Bit 4
BytesToRCSupportedFunctions.Byte18Bit04                := Bytes[18].4;
// Byte 18 - Bit 5
BytesToRCSupportedFunctions.Byte18Bit05                := Bytes[18].5;
// Byte 18 - Bit 6
BytesToRCSupportedFunctions.Byte18Bit06                := Bytes[18].6;
// Byte 18 - Bit 7
BytesToRCSupportedFunctions.Byte18Bit07                := Bytes[18].7;

END_FUNCTION

// Library/Functions/Convert/Misc/ByteToFragmentAction
FUNCTION ByteToFragmentAction : FragmentAction
// ------------------------------------------------------------------------- 
//  SRCI Robot Library                                                
// ------------------------------------------------------------------------- 
//                                                                           
//  Object:      FragmentActionToByte                                       
//  Author:      Thorsten Brach                                                
//  Date:        2024-11-05
//
//  Description:                                              
//   
//                                                                           
//  Copyright: 
//    (C) 2024 Thorsten Brach. All rights reserved                                                                                                                                            
//             Licensed under the LGPL-3.0 license.
//                                                                           
//  Disclaimer:                                                                           
//    This project is provided without any guarantee and can be used for   
//    private and commercial purposes. Any use is at the user’s 
//    own risk and responsibility.
//
// -------------------------------------------------------------------------
VAR_INPUT
  FragmentAction : BYTE;
END_VAR

ByteToFragmentAction.Complete:= FragmentAction.0; 
ByteToFragmentAction.Reset   := FragmentAction.1;   
ByteToFragmentAction.Clear   := FragmentAction.2;   
ByteToFragmentAction.BIT03   := FragmentAction.3;   
ByteToFragmentAction.BIT04   := FragmentAction.4;   
ByteToFragmentAction.BIT05   := FragmentAction.5;   
ByteToFragmentAction.BIT06   := FragmentAction.6;   
ByteToFragmentAction.BIT07   := FragmentAction.7;

END_FUNCTION

// Library/Functions/Convert/Misc/FragmentActionToByte
FUNCTION FragmentActionToByte : BYTE
// ------------------------------------------------------------------------- 
//  SRCI Robot Library                                                
// ------------------------------------------------------------------------- 
//                                                                           
//  Object:      FragmentActionToByte                                       
//  Author:      Thorsten Brach                                                
//  Date:        2024-06-01
//
//  Description:                                              
//   
//                                                                           
//  Copyright: 
//    (C) 2024 Thorsten Brach. All rights reserved                                                                                                                                            
//             Licensed under the LGPL-3.0 license.
//                                                                           
//  Disclaimer:                                                                           
//    This project is provided without any guarantee and can be used for   
//    private and commercial purposes. Any use is at the user’s 
//    own risk and responsibility.
//
// -------------------------------------------------------------------------
VAR_INPUT
  FragmentAction : FragmentAction;
END_VAR

FragmentActionToByte.0 := FragmentAction.Complete;
FragmentActionToByte.1 := FragmentAction.Reset;
FragmentActionToByte.2 := FragmentAction.Clear;
FragmentActionToByte.3 := FragmentAction.BIT03;
FragmentActionToByte.4 := FragmentAction.BIT04;
FragmentActionToByte.5 := FragmentAction.BIT05;
FragmentActionToByte.6 := FragmentAction.BIT06;
FragmentActionToByte.7 := FragmentAction.BIT07;

END_FUNCTION

// Library/Functions/Convert/Misc/ByteToVersion
FUNCTION ByteToVersion : VersionStruct
// ------------------------------------------------------------------------- 
//  SRCI Robot Library                                                
// ------------------------------------------------------------------------- 
//                                                                           
//  Object:      ByteToVersion                                       
//  Author:      Thorsten Brach                                                
//  Date:        2024-09-11
//
//  Description:                                              
//   
//                                                                           
//  Copyright: 
//    (C) 2024 Thorsten Brach. All rights reserved                                                                                                                                            
//             Licensed under the LGPL-3.0 license.
//                                                                           
//  Disclaimer:                                                                           
//    This project is provided without any guarantee and can be used for   
//    private and commercial purposes. Any use is at the user’s 
//    own risk and responsibility.
//
// -------------------------------------------------------------------------
VAR_INPUT
  /// Version
  Value : BYTE;
END_VAR

VAR
  _tmpByte : BYTE;
END_VAR

// Minor version  • Features
//                • 0..31 minor versions
ByteToVersion.MinorVersion.0 := Value.0;
ByteToVersion.MinorVersion.1 := Value.1;
ByteToVersion.MinorVersion.2 := Value.2;
ByteToVersion.MinorVersion.3 := Value.3;
ByteToVersion.MinorVersion.4 := Value.4;

// Major version  • Breaking change
//                • 0..7 major versions
ByteToVersion.MajorVersion.0 := Value.5;
ByteToVersion.MajorVersion.1 := Value.6;
ByteToVersion.MajorVersion.2 := Value.7;

END_FUNCTION

// Library/Functions/Convert/Misc/CombineBytesToUint
FUNCTION CombineBytesToUint : UINT
// ------------------------------------------------------------------------- 
//  SRCI Robot Library                                                
// ------------------------------------------------------------------------- 
//                                                                           
//  Object:      CombineBytes                                       
//  Author:      Thorsten Brach                                                
//  Date:        2024-09-03
//
//  Description:                                              
//   
//                                                                           
//  Copyright: 
//    (C) 2024 Thorsten Brach. All rights reserved                                                                                                                                            
//             Licensed under the LGPL-3.0 license.
//                                                                           
//  Disclaimer:                                                                           
//    This project is provided without any guarantee and can be used for   
//    private and commercial purposes. Any use is at the user’s 
//    own risk and responsibility.
//
// -------------------------------------------------------------------------
VAR_INPUT
  /// Byte to add as high byte
  HiByte : BYTE;
  /// Byte to add as low byte
  LoByte : BYTE;
END_VAR

CombineBytesToUint.0  := LoByte.0;
CombineBytesToUint.1  := LoByte.1;
CombineBytesToUint.2  := LoByte.2;
CombineBytesToUint.3  := LoByte.3;
CombineBytesToUint.4  := LoByte.4;
CombineBytesToUint.5  := LoByte.5;
CombineBytesToUint.6  := LoByte.6;
CombineBytesToUint.7  := LoByte.7;

CombineBytesToUint.8  := HiByte.0;
CombineBytesToUint.9  := HiByte.1;
CombineBytesToUint.10 := HiByte.2;
CombineBytesToUint.11 := HiByte.3;
CombineBytesToUint.12 := HiByte.4;
CombineBytesToUint.13 := HiByte.5;
CombineBytesToUint.14 := HiByte.6;
CombineBytesToUint.15 := HiByte.7;

END_FUNCTION

// Library/Functions/Convert/Misc/CombineHalfBytes
FUNCTION CombineHalfBytes : USINT
// ------------------------------------------------------------------------- 
//  SRCI Robot Library                                                
// ------------------------------------------------------------------------- 
//                                                                           
//  Object:      CombineHalfBytes                                       
//  Author:      Thorsten Brach                                                
//  Date:        2024-06-01
//
//  Description:                                              
//   
//                                                                           
//  Copyright: 
//    (C) 2024 Thorsten Brach. All rights reserved                                                                                                                                            
//             Licensed under the LGPL-3.0 license.
//                                                                           
//  Disclaimer:                                                                           
//    This project is provided without any guarantee and can be used for   
//    private and commercial purposes. Any use is at the user’s 
//    own risk and responsibility.
//
// -------------------------------------------------------------------------
VAR_INPUT
  /// Half-Byte to add to the upper 4 Bit
  HalfByteHi : BYTE;
  /// Half-Byte to add to the lower 4 Bit
  HalfByteLo : BYTE;
END_VAR

// merage ParSeq and Priority to combined variable
CombineHalfBytes.0 := HalfByteLo.0;
CombineHalfBytes.1 := HalfByteLo.1;
CombineHalfBytes.2 := HalfByteLo.2;
CombineHalfBytes.3 := HalfByteLo.3;

CombineHalfBytes.4 := HalfByteHi.0;
CombineHalfBytes.5 := HalfByteHi.1;
CombineHalfBytes.6 := HalfByteHi.2;
CombineHalfBytes.7 := HalfByteHi.3;

END_FUNCTION

// Library/Functions/Convert/Misc/CombineHalfSints
FUNCTION CombineHalfSints : USINT
// ------------------------------------------------------------------------- 
//  SRCI Robot Library                                                
// ------------------------------------------------------------------------- 
//                                                                           
//  Object:      CombineHalfSints                                       
//  Author:      Thorsten Brach                                                
//  Date:        2025-02-02
//
//  Description:                                              
//   
//                                                                           
//  Copyright: 
//    (C) 2025 Thorsten Brach. All rights reserved                                                                                                                                            
//             Licensed under the LGPL-3.0 license.
//                                                                           
//  Disclaimer:                                                                           
//    This project is provided without any guarantee and can be used for   
//    private and commercial purposes. Any use is at the user’s 
//    own risk and responsibility.
//
// -------------------------------------------------------------------------
VAR_INPUT
  /// Half-Sint to add to the upper 4 Bit
  HalfSintHi : SINT;
  /// Half-Sint to add to the lower 4 Bit
  HalfSintLo : SINT;
END_VAR

// merage ParSeq and Priority to combined variable
CombineHalfSints.0 := HalfSintLo.0;
CombineHalfSints.1 := HalfSintLo.1;
CombineHalfSints.2 := HalfSintLo.2;
CombineHalfSints.3 := HalfSintLo.3;

CombineHalfSints.4 := HalfSintHi.0;
CombineHalfSints.5 := HalfSintHi.1;
CombineHalfSints.6 := HalfSintHi.2;
CombineHalfSints.7 := HalfSintHi.3;

END_FUNCTION

// Library/Functions/Convert/Misc/DwordToRaStatusWord
FUNCTION DwordToRaStatusWord : RaStatusWord
// ------------------------------------------------------------------------- 
//  SRCI Robot Library                                                
// ------------------------------------------------------------------------- 
//                                                                           
//  Object:      DwordToRaStatusWord                                       
//  Author:      Thorsten Brach                                                
//  Date:        2024-11-16
//
//  Description:                                              
//   
//                                                                           
//  Copyright: 
//    (C) 2024 Thorsten Brach. All rights reserved                                                                                                                                            
//             Licensed under the LGPL-3.0 license.
//                                                                           
//  Disclaimer:                                                                           
//    This project is provided without any guarantee and can be used for   
//    private and commercial purposes. Any use is at the user’s 
//    own risk and responsibility.
//
// -------------------------------------------------------------------------
VAR_INPUT
  /// Value
  Value : DWORD;
END_VAR

DwordToRaStatusWord.IsMoving                 := Value.00;
DwordToRaStatusWord.PrimarySequencePaused    := Value.01;
DwordToRaStatusWord.InPrimaryPos             := Value.02;
DwordToRaStatusWord.SecondarySequenceActive  := Value.03;
DwordToRaStatusWord.IsBlending               := Value.04;
DwordToRaStatusWord.ErrorPending             := Value.05;
DwordToRaStatusWord.RestartInProgress        := Value.06;
DwordToRaStatusWord.Enabled                  := Value.07;
DwordToRaStatusWord.RaSequenceState.0        := Value.08;
DwordToRaStatusWord.RaSequenceState.1        := Value.09;
DwordToRaStatusWord.OperationMode.0          := Value.10;
DwordToRaStatusWord.OperationMode.1          := Value.11;
DwordToRaStatusWord.OperationMode.2          := Value.12;
DwordToRaStatusWord.CollisionDetectedEnabled := Value.13;
DwordToRaStatusWord.CollisionDetected        := Value.14;
DwordToRaStatusWord.RestartRequested         := Value.15;
DwordToRaStatusWord.Accelerating             := Value.16;
DwordToRaStatusWord.Decelerating             := Value.17;
DwordToRaStatusWord.ConstantVelocity         := Value.18;
DwordToRaStatusWord.Bit19                    := Value.19;
DwordToRaStatusWord.Bit20                    := Value.20;
DwordToRaStatusWord.Bit21                    := Value.21;
DwordToRaStatusWord.Bit22                    := Value.22;
DwordToRaStatusWord.Bit23                    := Value.23;
DwordToRaStatusWord.Bit24                    := Value.24;
DwordToRaStatusWord.Bit25                    := Value.25;
DwordToRaStatusWord.Bit26                    := Value.26;
DwordToRaStatusWord.Bit27                    := Value.27;
DwordToRaStatusWord.Bit28                    := Value.28;
DwordToRaStatusWord.Bit29                    := Value.29;
DwordToRaStatusWord.Bit30                    := Value.30;
DwordToRaStatusWord.Bit31                    := Value.31;

END_FUNCTION

// Library/Functions/Convert/Misc/PERCENT_INT_TO_REAL
FUNCTION PERCENT_INT_TO_REAL : REAL
// ------------------------------------------------------------------------- 
//  SRCI Robot Library                                                
// ------------------------------------------------------------------------- 
//                                                                           
//  Object:      PERCENT_INT_TO_REAL                                       
//  Author:      Thorsten Brach                                                
//  Date:        2025-02-07
//
//  Description:                                              
//   
//                                                                           
//  Copyright: 
//    (C) 2025 Thorsten Brach. All rights reserved                                                                                                                                            
//             Licensed under the LGPL-3.0 license.
//                                                                           
//  Disclaimer:                                                                           
//    This project is provided without any guarantee and can be used for   
//    private and commercial purposes. Any use is at the user’s 
//    own risk and responsibility.
//
// -------------------------------------------------------------------------
VAR_INPUT
  /// Percent value to convert 
  Value    : INT;
  /// value is an optional parameter ?  
  IsOptional : BOOL;
END_VAR

IF ( Value = 16#FFFF ) AND (IsOptional)// 16#FFFF for not supported values 
THEN
  PERCENT_INT_TO_REAL := -1.0;
  RETURN;
END_IF

PERCENT_INT_TO_REAL := INT_TO_REAL(Value) / RobotLibraryConstants.REAL_CONVERSION_FACTOR; {warning 'ToDo: check conversation is correct ?'}

END_FUNCTION

// Library/Functions/Convert/Misc/PlcOptionalCyclicToUint
FUNCTION PlcOptionalCyclicToUint : UINT
// ------------------------------------------------------------------------- 
//  SRCI Robot Library                                                
// ------------------------------------------------------------------------- 
//                                                                           
//  Object:      PlcOptionalCyclicToUint                                       
//  Author:      Thorsten Brach                                                
//  Date:        2024-11-30
//
//  Description:                                              
//   
//                                                                           
//  Copyright: 
//    (C) 2024 Thorsten Brach. All rights reserved                                                                                                                                            
//             Licensed under the LGPL-3.0 license.
//                                                                           
//  Disclaimer:                                                                           
//    This project is provided without any guarantee and can be used for   
//    private and commercial purposes. Any use is at the user’s 
//    own risk and responsibility.
//
// -------------------------------------------------------------------------
VAR_INPUT
  OptionalCyclic : AxesGroupParameterPlcOptionalCyclic;
END_VAR

PlcOptionalCyclicToUint.00 := OptionalCyclic.UseCallSubprogram;
PlcOptionalCyclicToUint.01 := OptionalCyclic.UseCartesianPosition;
PlcOptionalCyclicToUint.02 := OptionalCyclic.UseJointPosition;
PlcOptionalCyclicToUint.03 := OptionalCyclic.UseForce;
PlcOptionalCyclicToUint.04 := OptionalCyclic.Bit04;
PlcOptionalCyclicToUint.05 := OptionalCyclic.Bit05;
PlcOptionalCyclicToUint.06 := OptionalCyclic.Bit06;
PlcOptionalCyclicToUint.07 := OptionalCyclic.Bit07;  
PlcOptionalCyclicToUint.08 := OptionalCyclic.UseTwoSequences;
PlcOptionalCyclicToUint.09 := OptionalCyclic.UseCartesianPositionExt;
PlcOptionalCyclicToUint.10 := OptionalCyclic.UseJointPositionExt;
PlcOptionalCyclicToUint.11 := OptionalCyclic.Bit11;
PlcOptionalCyclicToUint.12 := OptionalCyclic.Bit12;
PlcOptionalCyclicToUint.13 := OptionalCyclic.Bit13;
PlcOptionalCyclicToUint.14 := OptionalCyclic.Bit14;
PlcOptionalCyclicToUint.15 := OptionalCyclic.Bit15;

END_FUNCTION

// Library/Functions/Convert/Misc/REAL_TO_PERCENT_INT
FUNCTION REAL_TO_PERCENT_INT : INT
// ------------------------------------------------------------------------- 
//  SRCI Robot Library                                                
// ------------------------------------------------------------------------- 
//                                                                           
//  Object:      REAL_TO_PERCENT_INT                                       
//  Author:      Thorsten Brach                                                
//  Date:        2025-02-07
//
//  Description:                                              
//   
//                                                                           
//  Copyright: 
//    (C) 2025 Thorsten Brach. All rights reserved                                                                                                                                            
//             Licensed under the LGPL-3.0 license.
//                                                                           
//  Disclaimer:                                                                           
//    This project is provided without any guarantee and can be used for   
//    private and commercial purposes. Any use is at the user’s 
//    own risk and responsibility.
//
// -------------------------------------------------------------------------
VAR_INPUT
  /// Percent value to convert 
  Value      : REAL;
  /// value is an optional parameter ?  
  IsOptional : BOOL;
END_VAR

IF ( Value = -1.0)  AND (IsOptional)// 16#FFFF for not supported values 
THEN
  REAL_TO_PERCENT_INT := UINT_TO_INT(16#FFFF);
  RETURN;
END_IF

REAL_TO_PERCENT_INT := REAL_TO_INT(Value * RobotLibraryConstants.REAL_CONVERSION_FACTOR);

END_FUNCTION

// Library/Functions/Convert/Misc/REAL_TO_PERCENT_UINT
FUNCTION REAL_TO_PERCENT_UINT : UINT
// ------------------------------------------------------------------------- 
//  SRCI Robot Library                                                
// ------------------------------------------------------------------------- 
//                                                                           
//  Object:      REAL_TO_PERCENT_UINT                                       
//  Author:      Thorsten Brach                                                
//  Date:        2025-02-07
//
//  Description:                                              
//   
//                                                                           
//  Copyright: 
//    (C) 2025 Thorsten Brach. All rights reserved                                                                                                                                            
//             Licensed under the LGPL-3.0 license.
//                                                                           
//  Disclaimer:                                                                           
//    This project is provided without any guarantee and can be used for   
//    private and commercial purposes. Any use is at the user’s 
//    own risk and responsibility.
//
// -------------------------------------------------------------------------
VAR_INPUT
  /// Percent value to convert 
  Value      : REAL;
  /// value is an optional parameter ?  
  IsOptional : BOOL;
END_VAR

IF ( Value = -1.0)  AND (IsOptional)// 16#FFFF for not supported values 
THEN
  REAL_TO_PERCENT_UINT := 16#FFFF;
  RETURN;
END_IF

REAL_TO_PERCENT_UINT := REAL_TO_UINT(Value * RobotLibraryConstants.REAL_CONVERSION_FACTOR);

END_FUNCTION

// Library/Functions/Convert/Misc/RobOptionalCyclicToUint
FUNCTION RobOptionalCyclicToUint : UINT
// ------------------------------------------------------------------------- 
//  SRCI Robot Library                                                
// ------------------------------------------------------------------------- 
//                                                                           
//  Object:      RobOptionalCyclicToUint                                       
//  Author:      Thorsten Brach                                                
//  Date:        2024-11-30
//
//  Description:                                              
//   
//                                                                           
//  Copyright: 
//    (C) 2024 Thorsten Brach. All rights reserved                                                                                                                                            
//             Licensed under the LGPL-3.0 license.
//                                                                           
//  Disclaimer:                                                                           
//    This project is provided without any guarantee and can be used for   
//    private and commercial purposes. Any use is at the user’s 
//    own risk and responsibility.
//
// -------------------------------------------------------------------------
VAR_INPUT
  OptionalCyclic : AxesGroupParameterRobOptionalCyclic;
END_VAR

RobOptionalCyclicToUint.00 := OptionalCyclic.UseCallSubprogram;      
RobOptionalCyclicToUint.01 := OptionalCyclic.UseCartesianPosition;   
RobOptionalCyclicToUint.02 := OptionalCyclic.UseJointPosition;       
RobOptionalCyclicToUint.03 := OptionalCyclic.UseForce;               
RobOptionalCyclicToUint.04 := OptionalCyclic.UseCurrent;             
RobOptionalCyclicToUint.05 := OptionalCyclic.Bit05;                  
RobOptionalCyclicToUint.06 := OptionalCyclic.Bit06;                  
RobOptionalCyclicToUint.07 := OptionalCyclic.Bit07;                  
RobOptionalCyclicToUint.08 := OptionalCyclic.UseTwoSequences;        
RobOptionalCyclicToUint.09 := OptionalCyclic.UseCartesianPositionExt;
RobOptionalCyclicToUint.10 := OptionalCyclic.UseJointPositionExt;    
RobOptionalCyclicToUint.11 := OptionalCyclic.UseForceExt;            
RobOptionalCyclicToUint.12 := OptionalCyclic.UseCurrentExt;          
RobOptionalCyclicToUint.13 := OptionalCyclic.Bit13;                  
RobOptionalCyclicToUint.14 := OptionalCyclic.Bit14;                  
RobOptionalCyclicToUint.15 := OptionalCyclic.Bit15;

END_FUNCTION

// Library/Functions/Convert/Misc/VersionToByte
FUNCTION VersionToByte : BYTE
// ------------------------------------------------------------------------- 
//  SRCI Robot Library                                                
// ------------------------------------------------------------------------- 
//                                                                           
//  Object:      VersionToByte                                       
//  Author:      Thorsten Brach                                                
//  Date:        2024-06-01
//
//  Description:                                              
//   
//                                                                           
//  Copyright: 
//    (C) 2024 Thorsten Brach. All rights reserved                                                                                                                                            
//             Licensed under the LGPL-3.0 license.
//                                                                           
//  Disclaimer:                                                                           
//    This project is provided without any guarantee and can be used for   
//    private and commercial purposes. Any use is at the user’s 
//    own risk and responsibility.
//
// -------------------------------------------------------------------------
VAR_INPUT
  /// Version
  Value : VersionStruct;
END_VAR

VAR
  _tmpByte : BYTE;
END_VAR

// Minor version  • Features
//                • 0..31 minor versions
VersionToByte.0 := Value.MinorVersion.0;
VersionToByte.1 := Value.MinorVersion.1;
VersionToByte.2 := Value.MinorVersion.2;
VersionToByte.3 := Value.MinorVersion.3;
VersionToByte.4 := Value.MinorVersion.4;

// Major version  • Breaking change
//                • 0..7 major versions
VersionToByte.5 := Value.MajorVersion.0;
VersionToByte.6 := Value.MajorVersion.1;
VersionToByte.7 := Value.MajorVersion.2;

END_FUNCTION

// Library/Functions/Convert/Misc/WordToArmConfigElbow
FUNCTION WordToArmConfigElbow : ArmConfigElbow
// ------------------------------------------------------------------------- 
//  SRCI Robot Library                                                
// ------------------------------------------------------------------------- 
//                                                                           
//  Object:      WordToArmConfigElbow                                       
//  Author:      Thorsten Brach                                                
//  Date:        2024-12-24
//
//  Description:                                              
//   
//                                                                           
//  Copyright: 
//    (C) 2024 Thorsten Brach. All rights reserved                                                                                                                                            
//             Licensed under the LGPL-3.0 license.
//                                                                           
//  Disclaimer:                                                                           
//    This project is provided without any guarantee and can be used for   
//    private and commercial purposes. Any use is at the user’s 
//    own risk and responsibility.
//
// -------------------------------------------------------------------------
VAR_INPUT
  /// Value
  Value : WORD;
END_VAR

VAR
  _tmpByte : BYTE;
END_VAR

IF (Value.1)
THEN
  WordToArmConfigElbow := ArmConfigElbow.DOWN;
ELSE
  WordToArmConfigElbow := ArmConfigElbow.UP;  
END_IF

END_FUNCTION

// Library/Functions/Convert/Misc/WordToArmConfigShoulder
FUNCTION WordToArmConfigShoulder : ArmConfigShoulder
// ------------------------------------------------------------------------- 
//  SRCI Robot Library                                                
// ------------------------------------------------------------------------- 
//                                                                           
//  Object:      WordToArmConfigShoulder                                       
//  Author:      Thorsten Brach                                                
//  Date:        2024-12-24
//
//  Description:                                              
//   
//                                                                           
//  Copyright: 
//    (C) 2024 Thorsten Brach. All rights reserved                                                                                                                                            
//             Licensed under the LGPL-3.0 license.
//                                                                           
//  Disclaimer:                                                                           
//    This project is provided without any guarantee and can be used for   
//    private and commercial purposes. Any use is at the user’s 
//    own risk and responsibility.
//
// -------------------------------------------------------------------------
VAR_INPUT
  /// Value
  Value : WORD;
END_VAR

VAR
  _tmpByte : BYTE;
END_VAR

IF (Value.0)
THEN
  WordToArmConfigShoulder := ArmConfigShoulder.BACK;
ELSE
  WordToArmConfigShoulder := ArmConfigShoulder.FRONT;  
END_IF

END_FUNCTION

// Library/Functions/Convert/Misc/WordToArmConfigWrist
FUNCTION WordToArmConfigWrist : ArmConfigWrist
// ------------------------------------------------------------------------- 
//  SRCI Robot Library                                                
// ------------------------------------------------------------------------- 
//                                                                           
//  Object:      WordToArmConfigWrist                                       
//  Author:      Thorsten Brach                                                
//  Date:        2024-12-24
//
//  Description:                                              
//   
//                                                                           
//  Copyright: 
//    (C) 2024 Thorsten Brach. All rights reserved                                                                                                                                            
//             Licensed under the LGPL-3.0 license.
//                                                                           
//  Disclaimer:                                                                           
//    This project is provided without any guarantee and can be used for   
//    private and commercial purposes. Any use is at the user’s 
//    own risk and responsibility.
//
// -------------------------------------------------------------------------
VAR_INPUT
  /// Value
  Value : WORD;
END_VAR

VAR
  _tmpByte : BYTE;
END_VAR

IF (Value.2)
THEN
  WordToArmConfigWrist := ArmConfigWrist.FLIP;
ELSE
  WordToArmConfigWrist := ArmConfigWrist.NON_FLIP;  
END_IF

END_FUNCTION

// Library/Functions/Convert/TO_STRING/AREA_TYPE_TO_STRING
FUNCTION AREA_TYPE_TO_STRING : STRING
// ------------------------------------------------------------------------- 
//  SRCI Robot Library                                                
// ------------------------------------------------------------------------- 
//                                                                           
//  Object:      AREA_TYPE_TO_STRING                                       
//  Author:      Thorsten Brach                                                
//  Date:        2025-02-01
//
//  Description:                                              
//   
//                                                                           
//  Copyright: 
//    (C) 2025 Thorsten Brach. All rights reserved                                                                                                                                            
//             Licensed under the LGPL-3.0 license.
//                                                                           
//  Disclaimer:                                                                           
//    This project is provided without any guarantee and can be used for   
//    private and commercial purposes. Any use is at the user’s 
//    own risk and responsibility.
//
// -------------------------------------------------------------------------
VAR_INPUT
  /// AreaType
  Value : AreaType;
END_VAR

CASE Value 
OF

  AreaType.AXES     : StrReplace('AXES ({0})'     ,'{0}' , USINT_TO_STRING(Value));
  AreaType.BOX      : StrReplace('BOX ({0})'      ,'{0}' , USINT_TO_STRING(Value));
  AreaType.CYLINDER : StrReplace('CYLINDER ({0})' ,'{0}' , USINT_TO_STRING(Value));
  AreaType.SPHERE   : StrReplace('SPHERE ({0})'   ,'{0}' , USINT_TO_STRING(Value));

END_CASE

END_FUNCTION

// Library/Functions/Convert/TO_STRING/ARM_CONFIG_ELBOW_TO_STRING
FUNCTION ARM_CONFIG_ELBOW_TO_STRING : STRING
// ------------------------------------------------------------------------- 
//  SRCI Robot Library                                                
// ------------------------------------------------------------------------- 
//                                                                           
//  Object:      ARM_CONFIG_ELBOW_TO_STRING                                       
//  Author:      Thorsten Brach                                                
//  Date:        2025-02-04
//
//  Description:                                              
//   
//                                                                           
//  Copyright: 
//    (C) 2025 Thorsten Brach. All rights reserved                                                                                                                                            
//             Licensed under the LGPL-3.0 license.
//                                                                           
//  Disclaimer:                                                                           
//    This project is provided without any guarantee and can be used for   
//    private and commercial purposes. Any use is at the user’s 
//    own risk and responsibility.
//
// -------------------------------------------------------------------------
VAR_INPUT
  /// ArmConfigElbow
  Value : ArmConfigElbow;
END_VAR

CASE Value 
OF

  ArmConfigElbow.USE_CONFIG : StrReplace('Elbow = USE_CONFIG ({0})','{0}' , INT_TO_STRING(Value));
  ArmConfigElbow.SAME       : StrReplace('Elbow = SAME ({0})'      ,'{0}' , INT_TO_STRING(Value));
  ArmConfigElbow.FREE       : StrReplace('Elbow = FREE ({0})'      ,'{0}' , INT_TO_STRING(Value));
  ArmConfigElbow.DOWN       : StrReplace('Elbow = DOWN ({0})'      ,'{0}' , INT_TO_STRING(Value));
  ArmConfigElbow.UP         : StrReplace('Elbow = UP ({0})'        ,'{0}' , INT_TO_STRING(Value));
  
END_CASE

END_FUNCTION

// Library/Functions/Convert/TO_STRING/ARM_CONFIG_SHOULDER_TO_STRING
FUNCTION ARM_CONFIG_SHOULDER_TO_STRING : STRING
// ------------------------------------------------------------------------- 
//  SRCI Robot Library                                                
// ------------------------------------------------------------------------- 
//                                                                           
//  Object:      ARM_CONFIG_SHOULDER_TO_STRING                                       
//  Author:      Thorsten Brach                                                
//  Date:        2025-02-04
//
//  Description:                                              
//   
//                                                                           
//  Copyright: 
//    (C) 2025 Thorsten Brach. All rights reserved                                                                                                                                            
//             Licensed under the LGPL-3.0 license.
//                                                                           
//  Disclaimer:                                                                           
//    This project is provided without any guarantee and can be used for   
//    private and commercial purposes. Any use is at the user’s 
//    own risk and responsibility.
//
// -------------------------------------------------------------------------
VAR_INPUT
  /// ArmConfigShoulder
  Value : ArmConfigShoulder;
END_VAR

CASE Value 
OF

  ArmConfigShoulder.USE_CONFIG : StrReplace('Shoulder = USE_CONFIG ({0})','{0}' , INT_TO_STRING(Value));
  ArmConfigShoulder.SAME       : StrReplace('Shoulder = SAME ({0})'      ,'{0}' , INT_TO_STRING(Value));
  ArmConfigShoulder.FREE       : StrReplace('Shoulder = FREE ({0})'      ,'{0}' , INT_TO_STRING(Value));
  ArmConfigShoulder.BACK       : StrReplace('Shoulder = BACK ({0})'      ,'{0}' , INT_TO_STRING(Value));
  ArmConfigShoulder.FRONT      : StrReplace('Shoulder = FRONT ({0})'     ,'{0}' , INT_TO_STRING(Value));
  
END_CASE

END_FUNCTION

// Library/Functions/Convert/TO_STRING/ARM_CONFIG_TO_STRING
FUNCTION ARM_CONFIG_TO_STRING : STRING
// ------------------------------------------------------------------------- 
//  SRCI Robot Library                                                
// ------------------------------------------------------------------------- 
//                                                                           
//  Object:      ARM_CONFIG_TO_STRING                                       
//  Author:      Thorsten Brach                                                
//  Date:        2025-01-23
//
//  Description:                                              
//   
//                                                                           
//  Copyright: 
//    (C) 2025 Thorsten Brach. All rights reserved                                                                                                                                            
//             Licensed under the LGPL-3.0 license.
//                                                                           
//  Disclaimer:                                                                           
//    This project is provided without any guarantee and can be used for   
//    private and commercial purposes. Any use is at the user’s 
//    own risk and responsibility.
//
// -------------------------------------------------------------------------
VAR_INPUT
  /// ArmConfigParameter
  Value : ArmConfigParameter;
END_VAR

VAR
  /// temporary byte
 _tmpByte : BYTE;
END_VAR

ARM_CONFIG_TO_STRING := '';
ARM_CONFIG_TO_STRING := CONCAT(ARM_CONFIG_TO_STRING , ARM_CONFIG_SHOULDER_TO_STRING(Value.Shoulder));
ARM_CONFIG_TO_STRING := CONCAT(ARM_CONFIG_TO_STRING ,' ; ');
ARM_CONFIG_TO_STRING := CONCAT(ARM_CONFIG_TO_STRING , ARM_CONFIG_ELBOW_TO_STRING(Value.Elbow));
ARM_CONFIG_TO_STRING := CONCAT(ARM_CONFIG_TO_STRING ,' ; ');
ARM_CONFIG_TO_STRING := CONCAT(ARM_CONFIG_TO_STRING , ARM_CONFIG_WRIST_TO_STRING(Value.Wrist));

END_FUNCTION

// Library/Functions/Convert/TO_STRING/ARM_CONFIG_WRIST_TO_STRING
FUNCTION ARM_CONFIG_WRIST_TO_STRING : STRING
// ------------------------------------------------------------------------- 
//  SRCI Robot Library                                                
// ------------------------------------------------------------------------- 
//                                                                           
//  Object:      ARM_CONFIG_WRIST_TO_STRING                                       
//  Author:      Thorsten Brach                                                
//  Date:        2025-02-04
//
//  Description:                                              
//   
//                                                                           
//  Copyright: 
//    (C) 2025 Thorsten Brach. All rights reserved                                                                                                                                            
//             Licensed under the LGPL-3.0 license.
//                                                                           
//  Disclaimer:                                                                           
//    This project is provided without any guarantee and can be used for   
//    private and commercial purposes. Any use is at the user’s 
//    own risk and responsibility.
//
// -------------------------------------------------------------------------
VAR_INPUT
  /// ArmConfigWrist
  Value : ArmConfigWrist;
END_VAR

CASE Value 
OF

  ArmConfigWrist.USE_CONFIG : StrReplace('Wrist = USE_CONFIG ({0})','{0}' , INT_TO_STRING(Value));
  ArmConfigWrist.SAME       : StrReplace('Wrist = SAME ({0})'      ,'{0}' , INT_TO_STRING(Value));
  ArmConfigWrist.FREE       : StrReplace('Wrist = FREE ({0})'      ,'{0}' , INT_TO_STRING(Value));
  ArmConfigWrist.FLIP       : StrReplace('Wrist = FLIP ({0})'      ,'{0}' , INT_TO_STRING(Value));
  ArmConfigWrist.NON_FLIP   : StrReplace('Wrist = NON_FLIP ({0})'  ,'{0}' , INT_TO_STRING(Value));

END_CASE

END_FUNCTION

// Library/Functions/Convert/TO_STRING/BLENDING_MODE_TO_STRING
FUNCTION BLENDING_MODE_TO_STRING : STRING
// ------------------------------------------------------------------------- 
//  SRCI Robot Library                                                
// ------------------------------------------------------------------------- 
//                                                                           
//  Object:      BLENDING_MODE_TO_STRING                                       
//  Author:      Thorsten Brach                                                
//  Date:        2025-01-23
//
//  Description:                                              
//   
//                                                                           
//  Copyright: 
//    (C) 2025 Thorsten Brach. All rights reserved                                                                                                                                            
//             Licensed under the LGPL-3.0 license.
//                                                                           
//  Disclaimer:                                                                           
//    This project is provided without any guarantee and can be used for   
//    private and commercial purposes. Any use is at the user’s 
//    own risk and responsibility.
//
// -------------------------------------------------------------------------
VAR_INPUT
  /// BlendingMode
  Value : BlendingMode;
END_VAR

CASE Value 
OF

